TYPE ST_MarkDefinition :
STRUCT
  nId : UDINT;        // mark id (array index)
  fHeight : REAL;     // triangle height (size Y)
  fLength : REAL;     // triangle lenght (size X)
  bInvertedX : BOOL;  // flipped in X axis (prior bMarksInverted)
  //bInvertedY : BOOL;  // flipped in Y axis
  fPosX : REAL;       // position X offset from 0/0
  fPosY : REAL;       // position > offset from 0/0
  sState : ST_MarkState;    // mark detection state
END_STRUCT 
END_TYPE

(* stored: Version 1.1.0.1, ProductVersion 3.1.4024.11
   DUT ST_MarkDefinition: Id {42950c73-347e-4e7c-859f-806b1921cf57} *)
